# EPICS substitutions: cpswAsynPortDriverApp/Db/test.substitutions
file driver_head.template
{
    pattern{ driver }
    { AxiXadc }
}

file driver_string.template
{
    pattern { NAME }
    { Temperature }
    { VccInt }
    { VccAux }
    { Vin }
    { VrefP }
    { VrefN }
    { VccBram }
    { SupplyOffsetA }
    { AdcOffsetA }
    { AdcGainA }
    { VccpInt }
    { VccpAux }
    { VccpDdr }
    { VinAux00 }
    { VinAux01 }
    { VinAux02 }
    { VinAux03 }
    { VinAux04 }
    { VinAux05 }
    { VinAux06 }
    { VinAux07 }
    { VinAux08 }
    { VinAux09 }
    { VinAux10 }
    { VinAux11 }
    { VinAux12 }
    { VinAux13 }
    { VinAux14 }
    { VinAux15 }
    { TemperatureMax  }
    { VccIntMax }
    { VccAuxMax }
    { VccBramMax }
    { TemperatureMin }
    { VccIntMin }
    { VccAuxMin }
    { VccBramMin }
    { VccpIntMax }
    { VccpAuxMax }
    { VccpDdrMax }
    { VccpIntMin }
    { VccpAuxMin }
    { VccpDdrMin }
    { Flag }
    { VccpIntMax }
}
file driver_tail.template
{
    pattern{ driver }
    { AxiXadc }
}
file driver_param.template
{
   pattern { NAME }
    { Temperature }
    { VccInt }
    { VccAux }
    { Vin }
    { VrefP }
    { VrefN }
    { VccBram }
    { SupplyOffsetA }
    { AdcOffsetA }
    { AdcGainA }
    { VccpInt }
    { VccpAux }
    { VccpDdr }
    { VinAux00 }
    { VinAux01 }
    { VinAux02 }
    { VinAux03 }
    { VinAux04 }
    { VinAux05 }
    { VinAux06 }
    { VinAux07 }
    { VinAux08 }
    { VinAux09 }
    { VinAux10 }
    { VinAux11 }
    { VinAux12 }
    { VinAux13 }
    { VinAux14 }
    { VinAux15 }
    { TemperatureMax  }
    { VccIntMax }
    { VccAuxMax }
    { VccBramMax }
    { TemperatureMin }
    { VccIntMin }
    { VccAuxMin }
    { VccBramMin }
    { VccpIntMax }
    { VccpAuxMax }
    { VccpDdrMax }
    { VccpIntMin }
    { VccpAuxMin }
    { VccpDdrMin }
    { Flag }
}
